(* PLC project sensor_fault, Dassault Systèmes ControlBuild 2024x *)
(* stored: creationDateTime 2023-10-03T11:12:54-01:00 *)

(* This module makes it possible to generate faults on sensors (actors/products) thanks to graphical interface. It is not an actor. *)
FUNCTION_BLOCK equipment_library.sensor_fault
  VAR_INPUT
    sensorVal : BOOL := false;
  END_VAR
  VAR_OUTPUT
    val : BOOL := false;
  END_VAR
  VAR
    d_sensor : BOOL := false;
    v_d_sensor : BOOL := false;
  END_VAR


ACTION C_source_code:
/* ----------------------------------------------------------------	*/
/* Type : Model of Operative Behaviour					*/
/* Category :  Actors and Products						*/
/* Author : Dassault Systemes						*/
/* Update date : June 2018							*/
/* ----------------------------------------------------------------	*/
/* This module makes it possible to generate faults on sensors 	*/
/* (actors/products) thanks to graphical interface.			*/
/* It is not an actor.							*/
/* ----------------------------------------------------------------	*/

if (d_sensor) val = v_d_sensor;
 else val = sensorVal;
END_ACTION
END_FUNCTION_BLOCK
